(* Logix 5000 project; controller L3 vendor 1 type 14 code 92 rev 20.12; software revision 20.04; part 2 of 9 *)
(* tags used below, declared in another part *)
   B3 : DINT[100];
   CONV_PID_N10_170 : PID;   // *** Tag created for conversion to PID type required for instruction translation ***
   CV_PID_wkk : DINT;
   cv_pmpano : DINT;
   cv_pmprenv : DINT;
   DateTime : DINT[7];   // DINT array tag for retrieve wallclock time through GSV created during conversion
   dbpmpeau : DINT;
   def_ready_pmp_decap_1 : BOOL;
   def_ready_pmp_decap_2 : BOOL;
   def_ready_pmpeau1 : BOOL;
   def_ready_pmpeau2 : BOOL;
   def_ready_ventilo_eau_1 : BOOL;
   def_ready_ventilo_eau_2 : BOOL;
   def_ready_ventilo_eau_3 : BOOL;
   dmd_run_pmp1_decap : BOOL;
   dmd_run_pmp2_decap : BOOL;
   F8 : REAL[100];
   L3_stat : DINT[20];
   limb_pmpeau : DINT;
   limh_pmpeau : DINT;
   N10 : DINT[233];
   N20 : DINT[200];
   N7 : DINT[200];
   N9 : DINT[200];   // niveau decapage vers lancy (n9[10) ;;N9[70]
   ok_arm_io_decap : BOOL;
   okpmpeau1 : BOOL;
   okpmpeau2 : BOOL;
   okventilotour1 : BOOL;
   okventilotour2 : BOOL;
   okventilotour3 : BOOL;
   pid_ANO : PID;
   pid_colmat : PID;
   pid_deg : PID;
   pid_pmpANO : PID;
   pid_pmprenvoi : PID;
   PIDwkk : PID;
   pmpano_inhold : BOOL;
   pmpano_inholdval : DINT;
   pmprenv_inhold : BOOL;
   pmprenv_inholdval : DINT;
   S_bP_dmd_man_pmp_eau : BOOL;
   s_bp_stop_soude : BOOL;
   s_bp_strt_soude : BOOL;
   s_csg_ventilo_ano : DINT;
   S_def_pmp_decap_1 : BOOL;
   S_def_pmp_decap_2 : BOOL;
   S_def_pmpeauano1 : BOOL;
   S_def_pmpeauano2 : BOOL;
   S_def_ventilo_eau1 : BOOL;
   S_def_ventilo_eau2 : BOOL;
   S_def_ventilo_eau3 : BOOL;
   S_FLOW_RETURN_LANCY : DINT;
   S_hiver : BOOL;
   s_nbr_ventilo_ano : DINT;
   S_Q_DEM_NAOH : DINT;
   S_RUN_PMP_DEC1 : BOOL;
   S_RUN_PMP_DEC2 : BOOL;
   S_run_pmpeauano1 : BOOL;
   S_run_pmpeauano2 : BOOL;
   S_run_ventilo_1 : BOOL;
   s_run_ventilo_2 : BOOL;
   S_run_ventilo_3 : BOOL;
   S_SPEED : DINT;
   S_T_ANO : DINT;
   scp_pmp_decap_1 : SCP;
   scp_pmp_decap_2 : SCP;
   scp_ventilo : SCP;
   stat_L3 : DINT[20];
   T4 : TIMER[180];
   T_man_pmp_eau : TIMER;
   T_pmp_decap_1 : TIMER;
   T_pmp_decap_2 : TIMER;
   T_pmpeau_1 : TIMER;
   T_pmpeau_2 : TIMER;
   T_ventilo_eau_1 : TIMER;
   T_ventilo_eau_2 : TIMER;
   T_ventilo_eau_3 : TIMER;
   TIE_PID_wkk : DINT;
   vit_pmp_dec_1 : REAL;
   vit_pmp_dec_2 : DINT;
   vit_renvoi_lancy : DINT;
   vit_ventilo : DINT;
   vitpmpeau : DINT;

PROGRAM _11_PID2   (* main routine _11_PID2 *)

ROUTINE _11_PID2   (* ladder *)
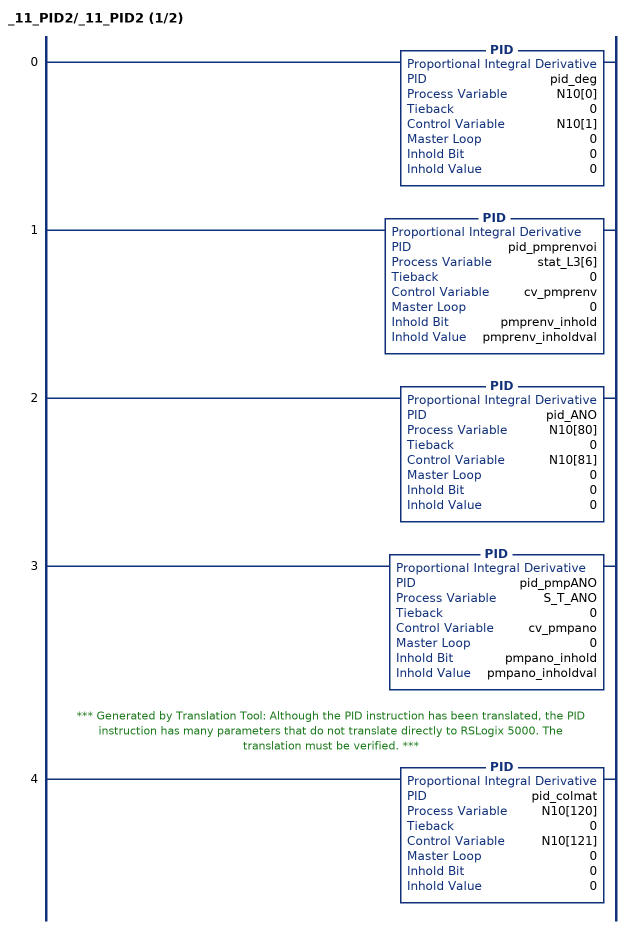
   0: PID(pid_deg,N10[0],0,N10[1],0,0,0);
   1: PID(pid_pmprenvoi,stat_L3[6],0,cv_pmprenv,0,pmprenv_inhold,pmprenv_inholdval);
   2: PID(pid_ANO,N10[80],0,N10[81],0,0,0);
   3: PID(pid_pmpANO,S_T_ANO,0,cv_pmpano,0,pmpano_inhold,pmpano_inholdval);
   // *** Generated by Translation Tool: Although the PID instruction has been translated, the PID instruction has many parameters that do not translate directly to RSLogix 5000. The translation must be verified. ***
   4: PID(pid_colmat,N10[120],0,N10[121],0,0,0);
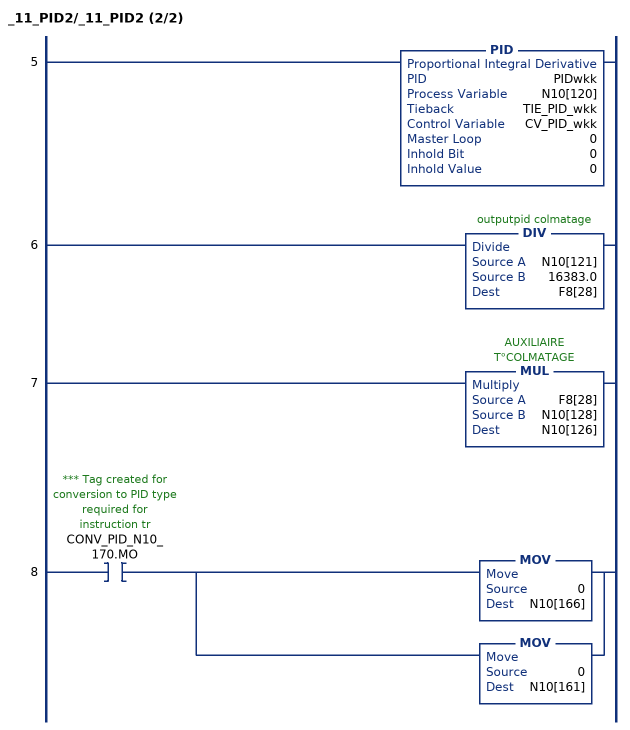
   5: PID(PIDwkk,N10[120],TIE_PID_wkk,CV_PID_wkk,0,0,0);
   6: DIV(N10[121],16383.0,F8[28]);
   7: MUL(F8[28],N10[128],N10[126]);
   8: XIC(CONV_PID_N10_170.MO)[MOV(0,N10[166]) ,MOV(0,N10[161]) ];
END_ROUTINE
END_PROGRAM

PROGRAM _2_GENERAL   (* main routine _2_GENERAL *)

ROUTINE _10_soude_conduct_tour   (* ladder *)
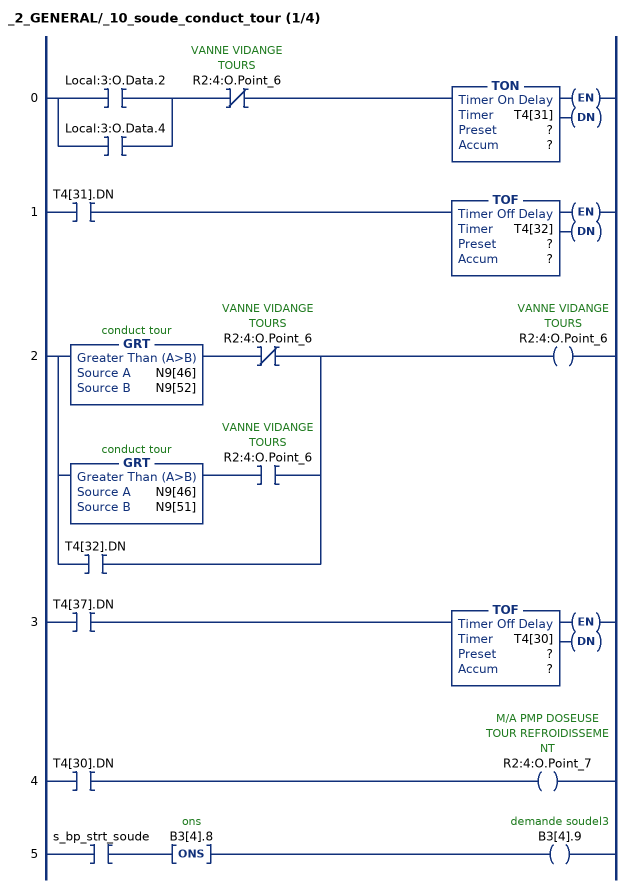
   0: [XIC(Local:3:O.Data.2) ,XIC(Local:3:O.Data.4) ]XIO(R2:4:O.Point_6)TON(T4[31],?,?);
   1: XIC(T4[31].DN)TOF(T4[32],?,?);
   2: [GRT(N9[46],N9[52]) XIO(R2:4:O.Point_6) ,GRT(N9[46],N9[51]) XIC(R2:4:O.Point_6) ,XIC(T4[32].DN) ]OTE(R2:4:O.Point_6);
   3: XIC(T4[37].DN)TOF(T4[30],?,?);
   4: XIC(T4[30].DN)OTE(R2:4:O.Point_7);
   5: XIC(s_bp_strt_soude)ONS(B3[4].8)OTE(B3[4].9);
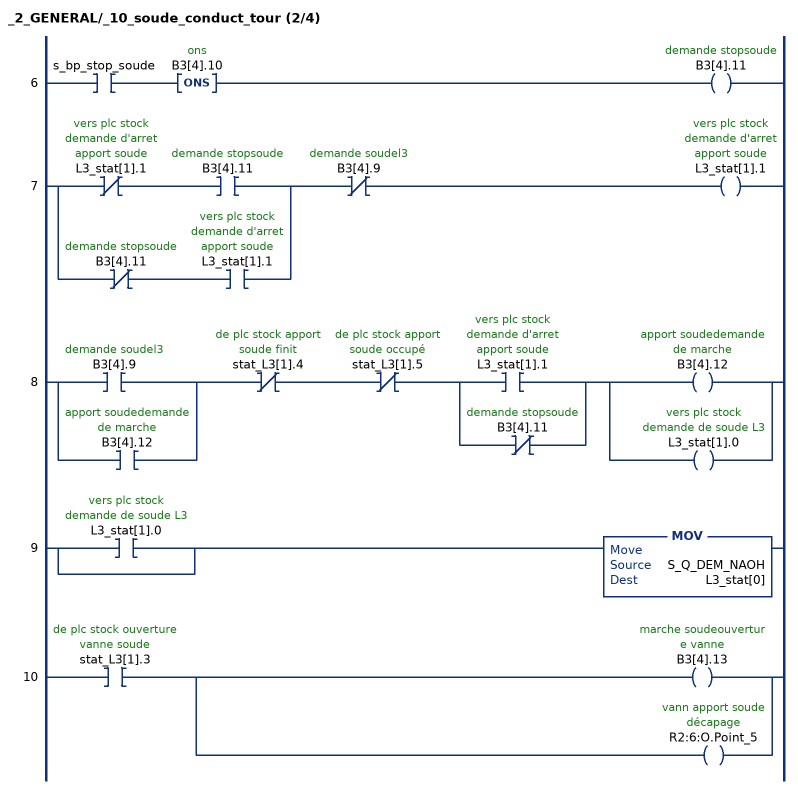
   6: XIC(s_bp_stop_soude)ONS(B3[4].10)OTE(B3[4].11);
   7: [XIO(L3_stat[1].1) XIC(B3[4].11) ,XIO(B3[4].11) XIC(L3_stat[1].1) ]XIO(B3[4].9)OTE(L3_stat[1].1);
   8: [XIC(B3[4].9) ,XIC(B3[4].12) ]XIO(stat_L3[1].4)XIO(stat_L3[1].5)[XIC(L3_stat[1].1) ,XIO(B3[4].11) ][OTE(B3[4].12) ,OTE(L3_stat[1].0) ];
   9: [XIC(L3_stat[1].0) ,]MOV(S_Q_DEM_NAOH,L3_stat[0]);
   10: XIC(stat_L3[1].3)[OTE(B3[4].13) ,OTE(R2:6:O.Point_5) ];
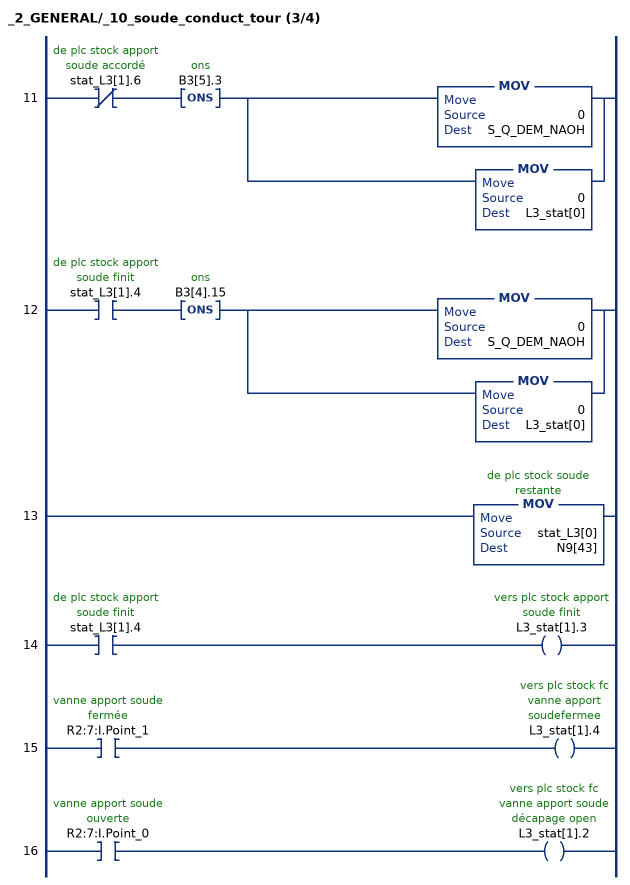
   11: XIO(stat_L3[1].6)ONS(B3[5].3)[MOV(0,S_Q_DEM_NAOH) ,MOV(0,L3_stat[0]) ];
   12: XIC(stat_L3[1].4)ONS(B3[4].15)[MOV(0,S_Q_DEM_NAOH) ,MOV(0,L3_stat[0]) ];
   13: MOV(stat_L3[0],N9[43]);
   14: XIC(stat_L3[1].4)OTE(L3_stat[1].3);
   15: XIC(R2:7:I.Point_1)OTE(L3_stat[1].4);
   16: XIC(R2:7:I.Point_0)OTE(L3_stat[1].2);
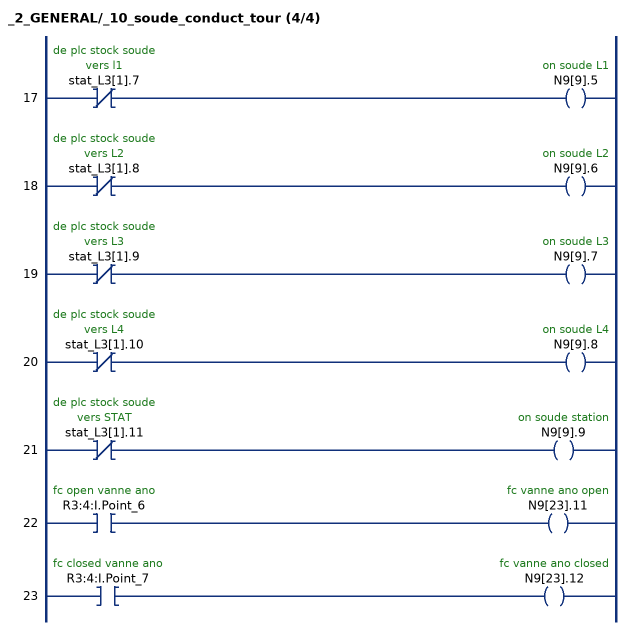
   17: XIO(stat_L3[1].7)OTE(N9[9].5);
   18: XIO(stat_L3[1].8)OTE(N9[9].6);
   19: XIO(stat_L3[1].9)OTE(N9[9].7);
   20: XIO(stat_L3[1].10)OTE(N9[9].8);
   21: XIO(stat_L3[1].11)OTE(N9[9].9);
   22: XIC(R3:4:I.Point_6)OTE(N9[23].11);
   23: XIC(R3:4:I.Point_7)OTE(N9[23].12);
END_ROUTINE

ROUTINE _11_pmp_eau_tour   (* ladder *)
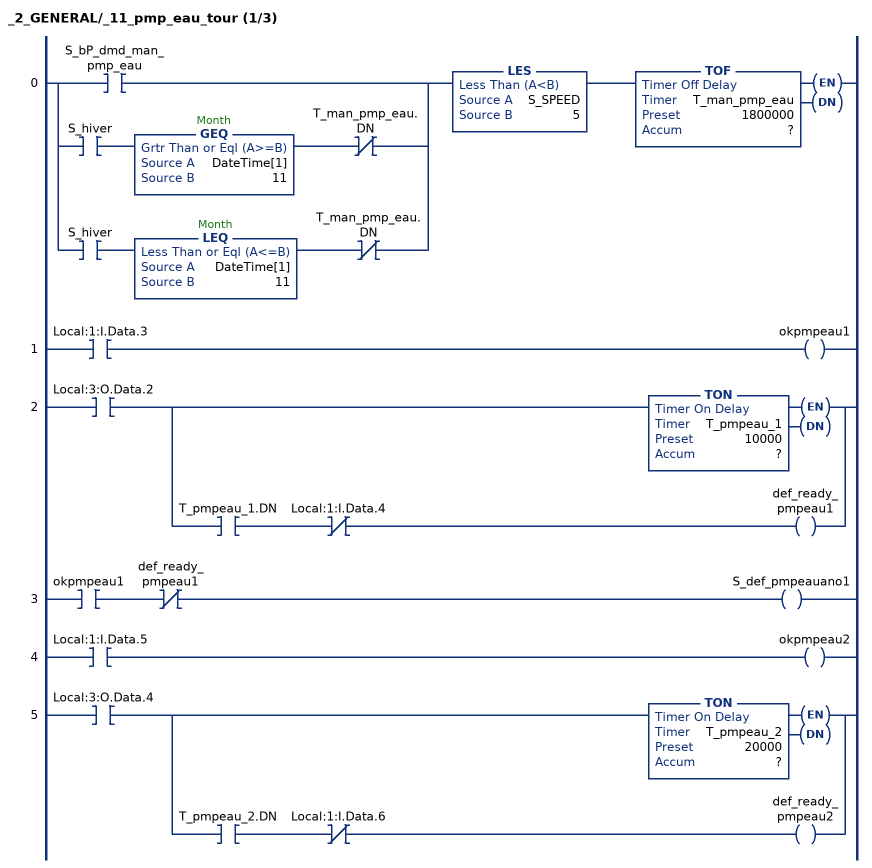
   0: [XIC(S_bP_dmd_man_pmp_eau) ,XIC(S_hiver) GEQ(DateTime[1],11) XIO(T_man_pmp_eau.DN) ,XIC(S_hiver) LEQ(DateTime[1],11) XIO(T_man_pmp_eau.DN) ]LES(S_SPEED,5)TOF(T_man_pmp_eau,?,?);
   1: XIC(Local:1:I.Data.3)OTE(okpmpeau1);
   2: XIC(Local:3:O.Data.2)[TON(T_pmpeau_1,?,?) ,XIC(T_pmpeau_1.DN) XIO(Local:1:I.Data.4) OTE(def_ready_pmpeau1) ];
   3: XIC(okpmpeau1)XIO(def_ready_pmpeau1)OTE(S_def_pmpeauano1);
   4: XIC(Local:1:I.Data.5)OTE(okpmpeau2);
   5: XIC(Local:3:O.Data.4)[TON(T_pmpeau_2,?,?) ,XIC(T_pmpeau_2.DN) XIO(Local:1:I.Data.6) OTE(def_ready_pmpeau2) ];
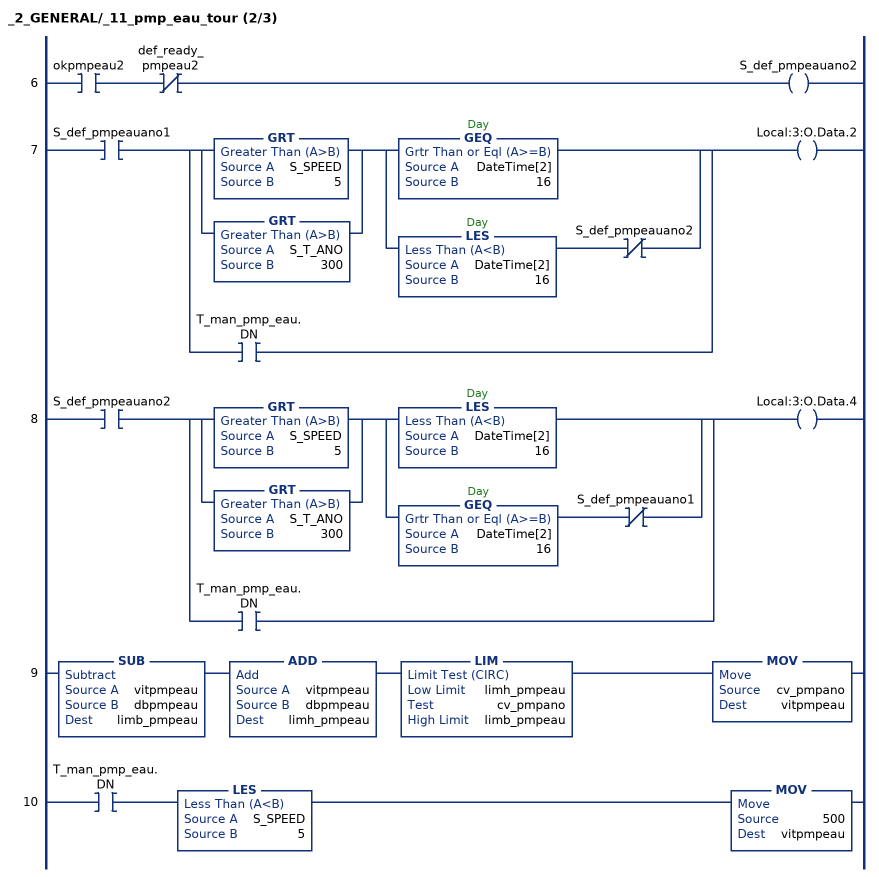
   6: XIC(okpmpeau2)XIO(def_ready_pmpeau2)OTE(S_def_pmpeauano2);
   7: XIC(S_def_pmpeauano1)[[GRT(S_SPEED,5) ,GRT(S_T_ANO,300) ] [GEQ(DateTime[2],16) ,LES(DateTime[2],16) XIO(S_def_pmpeauano2) ] ,XIC(T_man_pmp_eau.DN) ]OTE(Local:3:O.Data.2);
   8: XIC(S_def_pmpeauano2)[[GRT(S_SPEED,5) ,GRT(S_T_ANO,300) ] [LES(DateTime[2],16) ,GEQ(DateTime[2],16) XIO(S_def_pmpeauano1) ] ,XIC(T_man_pmp_eau.DN) ]OTE(Local:3:O.Data.4);
   9: SUB(vitpmpeau,dbpmpeau,limb_pmpeau)ADD(vitpmpeau,dbpmpeau,limh_pmpeau)LIM(limh_pmpeau,cv_pmpano,limb_pmpeau)MOV(cv_pmpano,vitpmpeau);
   10: XIC(T_man_pmp_eau.DN)LES(S_SPEED,5)MOV(500,vitpmpeau);
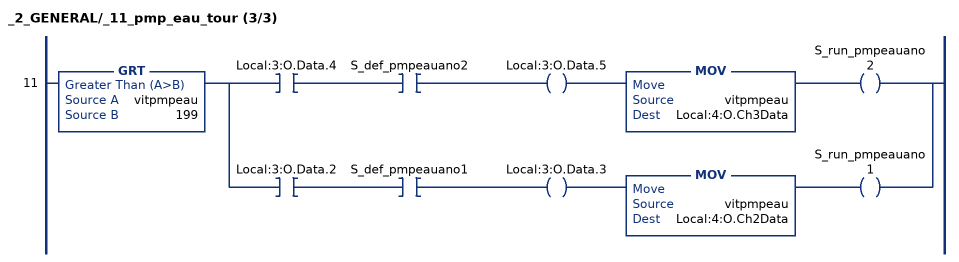
   11: GRT(vitpmpeau,199)[XIC(Local:3:O.Data.4) XIC(S_def_pmpeauano2) OTE(Local:3:O.Data.5) MOV(vitpmpeau,Local:4:O.Ch3Data) OTE(S_run_pmpeauano2) ,XIC(Local:3:O.Data.2) XIC(S_def_pmpeauano1) OTE(Local:3:O.Data.3) MOV(vitpmpeau,Local:4:O.Ch2Data) OTE(S_run_pmpeauano1) ];
END_ROUTINE

ROUTINE _12_ventilo_tour   (* ladder *)
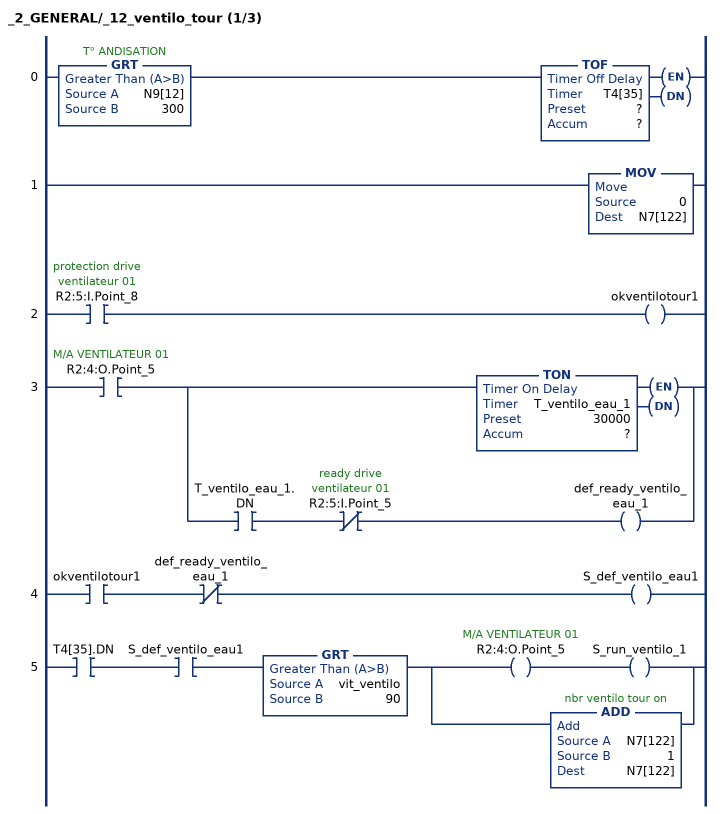
   0: GRT(N9[12],300)TOF(T4[35],?,?);
   1: MOV(0,N7[122]);
   2: XIC(R2:5:I.Point_8)OTE(okventilotour1);
   3: XIC(R2:4:O.Point_5)[TON(T_ventilo_eau_1,?,?) ,XIC(T_ventilo_eau_1.DN) XIO(R2:5:I.Point_5) OTE(def_ready_ventilo_eau_1) ];
   4: XIC(okventilotour1)XIO(def_ready_ventilo_eau_1)OTE(S_def_ventilo_eau1);
   5: XIC(T4[35].DN)XIC(S_def_ventilo_eau1)GRT(vit_ventilo,90)[OTE(R2:4:O.Point_5) OTE(S_run_ventilo_1) ,ADD(N7[122],1,N7[122]) ];
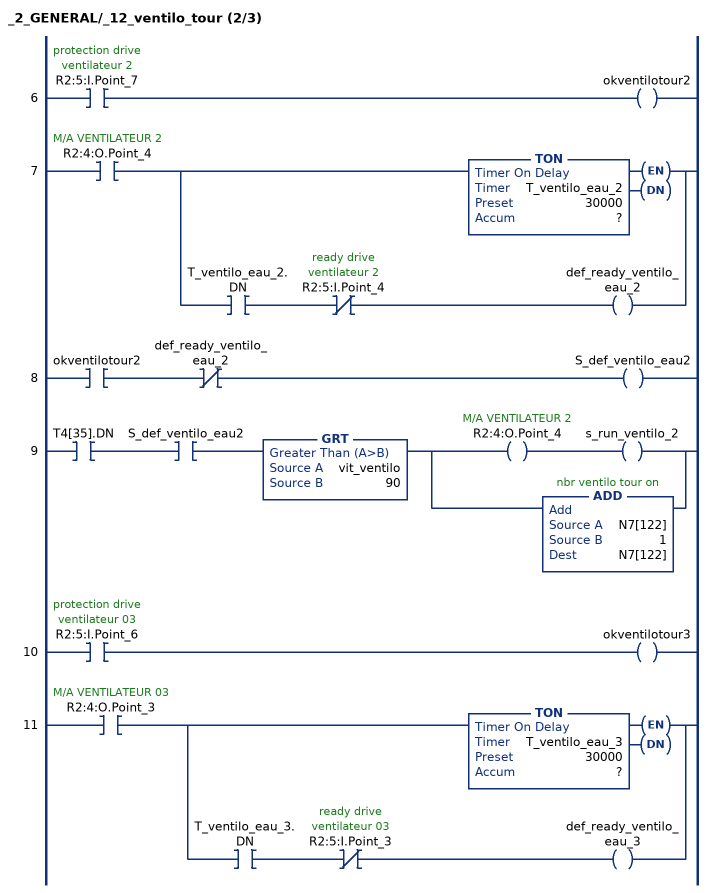
   6: XIC(R2:5:I.Point_7)OTE(okventilotour2);
   7: XIC(R2:4:O.Point_4)[TON(T_ventilo_eau_2,?,?) ,XIC(T_ventilo_eau_2.DN) XIO(R2:5:I.Point_4) OTE(def_ready_ventilo_eau_2) ];
   8: XIC(okventilotour2)XIO(def_ready_ventilo_eau_2)OTE(S_def_ventilo_eau2);
   9: XIC(T4[35].DN)XIC(S_def_ventilo_eau2)GRT(vit_ventilo,90)[OTE(R2:4:O.Point_4) OTE(s_run_ventilo_2) ,ADD(N7[122],1,N7[122]) ];
   10: XIC(R2:5:I.Point_6)OTE(okventilotour3);
   11: XIC(R2:4:O.Point_3)[TON(T_ventilo_eau_3,?,?) ,XIC(T_ventilo_eau_3.DN) XIO(R2:5:I.Point_3) OTE(def_ready_ventilo_eau_3) ];
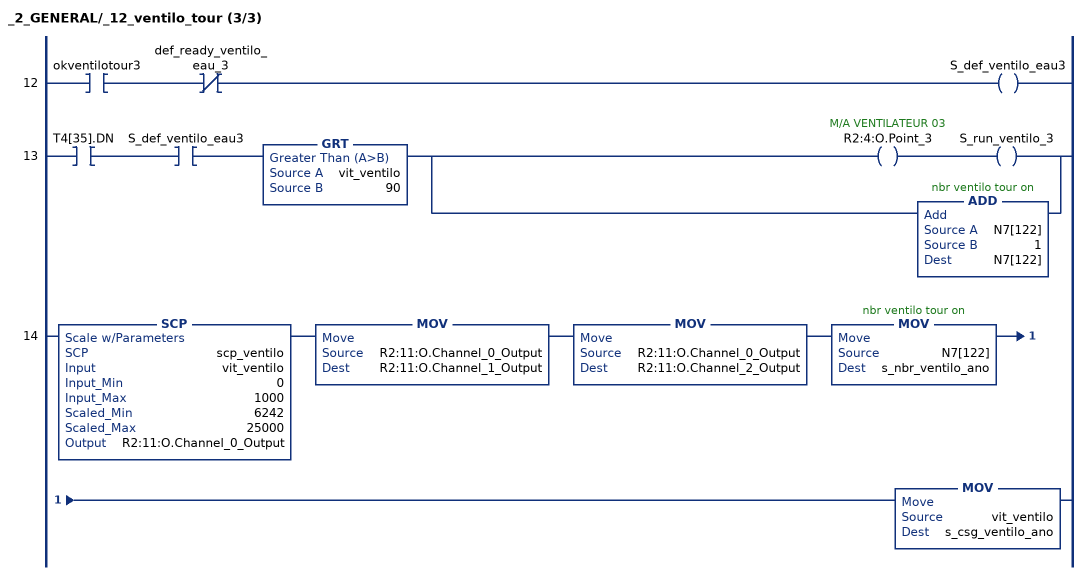
   12: XIC(okventilotour3)XIO(def_ready_ventilo_eau_3)OTE(S_def_ventilo_eau3);
   13: XIC(T4[35].DN)XIC(S_def_ventilo_eau3)GRT(vit_ventilo,90)[OTE(R2:4:O.Point_3) OTE(S_run_ventilo_3) ,ADD(N7[122],1,N7[122]) ];
   14: SCP(scp_ventilo,vit_ventilo,0,1000,6242,25000,R2:11:O.Channel_0_Output)MOV(R2:11:O.Channel_0_Output,R2:11:O.Channel_1_Output)MOV(R2:11:O.Channel_0_Output,R2:11:O.Channel_2_Output)MOV(N7[122],s_nbr_ventilo_ano)MOV(vit_ventilo,s_csg_ventilo_ano);
END_ROUTINE

ROUTINE _13_pmp_decap   (* ladder *)
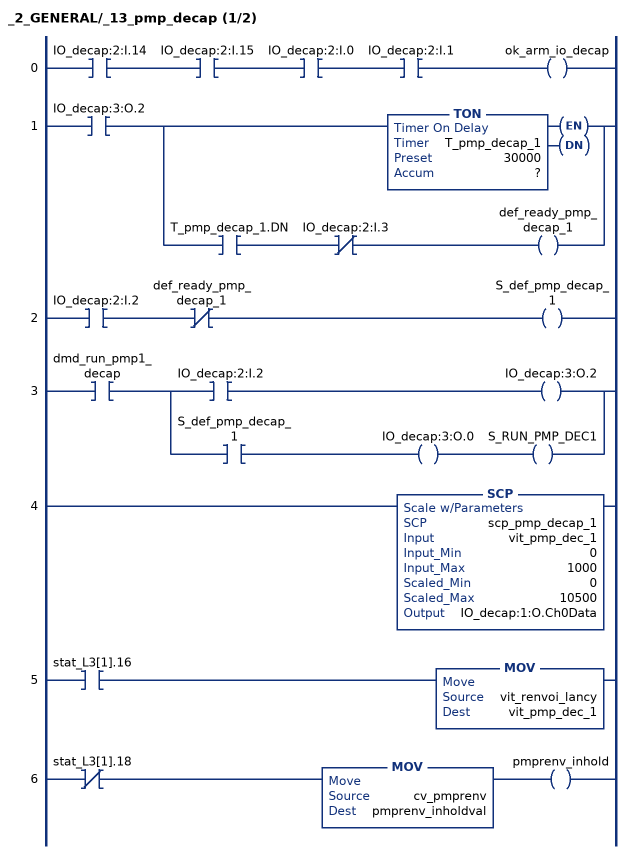
   0: XIC(IO_decap:2:I.14)XIC(IO_decap:2:I.15)XIC(IO_decap:2:I.0)XIC(IO_decap:2:I.1)OTE(ok_arm_io_decap);
   1: XIC(IO_decap:3:O.2)[TON(T_pmp_decap_1,?,?) ,XIC(T_pmp_decap_1.DN) XIO(IO_decap:2:I.3) OTE(def_ready_pmp_decap_1) ];
   2: XIC(IO_decap:2:I.2)XIO(def_ready_pmp_decap_1)OTE(S_def_pmp_decap_1);
   3: XIC(dmd_run_pmp1_decap)[XIC(IO_decap:2:I.2) OTE(IO_decap:3:O.2) ,XIC(S_def_pmp_decap_1) OTE(IO_decap:3:O.0) OTE(S_RUN_PMP_DEC1) ];
   4: SCP(scp_pmp_decap_1,vit_pmp_dec_1,0,1000,0,10500,IO_decap:1:O.Ch0Data);
   5: XIC(stat_L3[1].16)MOV(vit_renvoi_lancy,vit_pmp_dec_1);
   6: XIO(stat_L3[1].18)MOV(cv_pmprenv,pmprenv_inholdval)OTE(pmprenv_inhold);
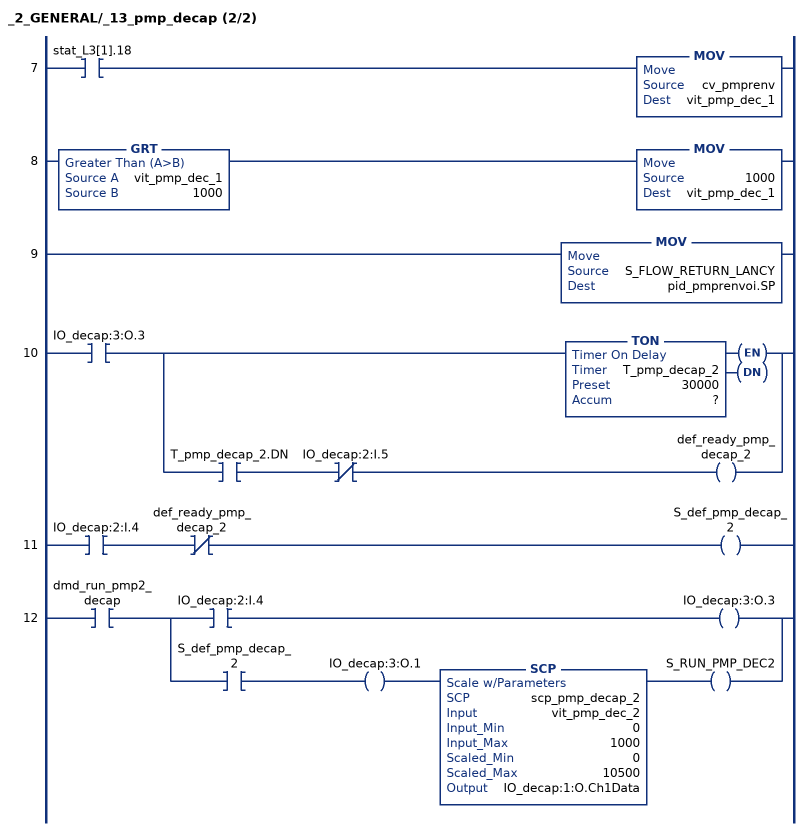
   7: XIC(stat_L3[1].18)MOV(cv_pmprenv,vit_pmp_dec_1);
   8: GRT(vit_pmp_dec_1,1000)MOV(1000,vit_pmp_dec_1);
   9: MOV(S_FLOW_RETURN_LANCY,pid_pmprenvoi.SP);
   10: XIC(IO_decap:3:O.3)[TON(T_pmp_decap_2,?,?) ,XIC(T_pmp_decap_2.DN) XIO(IO_decap:2:I.5) OTE(def_ready_pmp_decap_2) ];
   11: XIC(IO_decap:2:I.4)XIO(def_ready_pmp_decap_2)OTE(S_def_pmp_decap_2);
   12: XIC(dmd_run_pmp2_decap)[XIC(IO_decap:2:I.4) OTE(IO_decap:3:O.3) ,XIC(S_def_pmp_decap_2) OTE(IO_decap:3:O.1) SCP(scp_pmp_decap_2,vit_pmp_dec_2,0,1000,0,10500,IO_decap:1:O.Ch1Data) OTE(S_RUN_PMP_DEC2) ];
END_ROUTINE

ROUTINE _20_ALARM   (* ladder *)
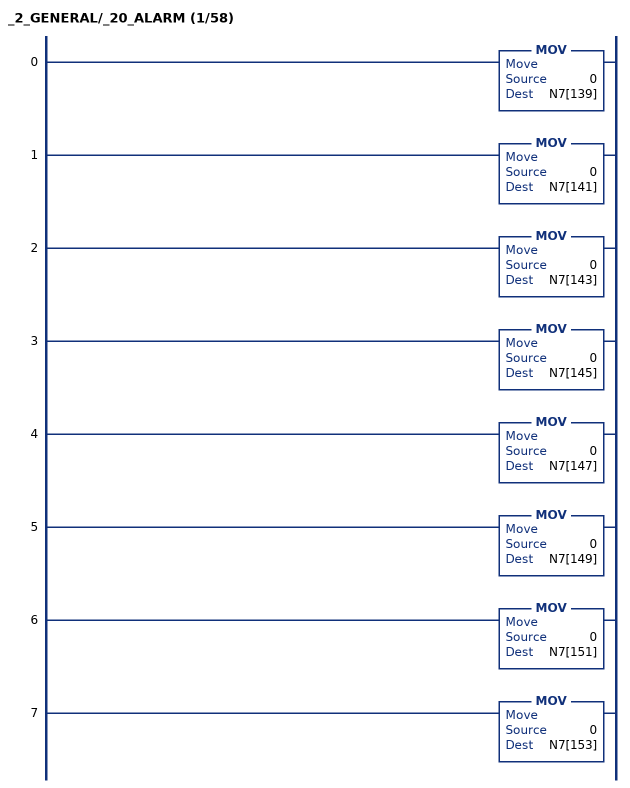
   0: MOV(0,N7[139]);
   1: MOV(0,N7[141]);
   2: MOV(0,N7[143]);
   3: MOV(0,N7[145]);
   4: MOV(0,N7[147]);
   5: MOV(0,N7[149]);
   6: MOV(0,N7[151]);
   7: MOV(0,N7[153]);
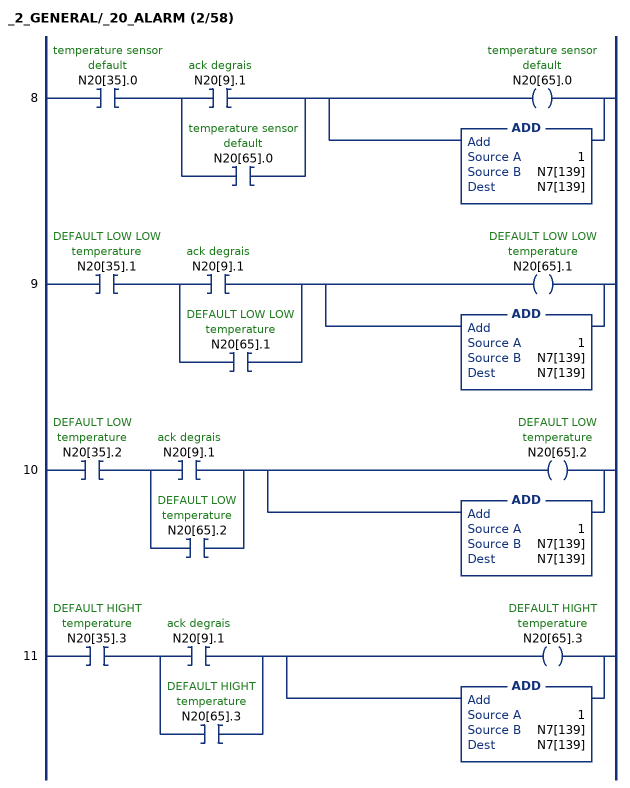
   8: XIC(N20[35].0)[XIC(N20[9].1) ,XIC(N20[65].0) ][OTE(N20[65].0) ,ADD(1,N7[139],N7[139]) ];
   9: XIC(N20[35].1)[XIC(N20[9].1) ,XIC(N20[65].1) ][OTE(N20[65].1) ,ADD(1,N7[139],N7[139]) ];
   10: XIC(N20[35].2)[XIC(N20[9].1) ,XIC(N20[65].2) ][OTE(N20[65].2) ,ADD(1,N7[139],N7[139]) ];
   11: XIC(N20[35].3)[XIC(N20[9].1) ,XIC(N20[65].3) ][OTE(N20[65].3) ,ADD(1,N7[139],N7[139]) ];
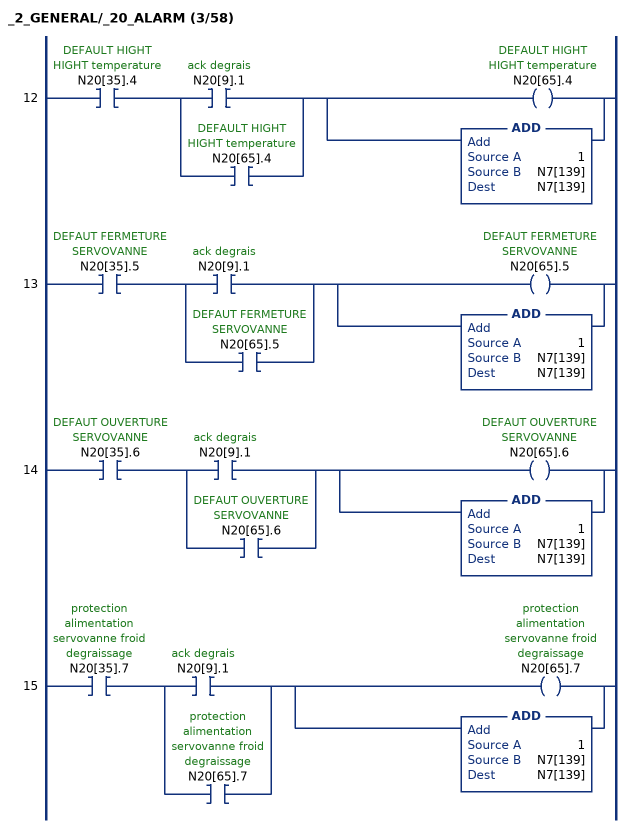
   12: XIC(N20[35].4)[XIC(N20[9].1) ,XIC(N20[65].4) ][OTE(N20[65].4) ,ADD(1,N7[139],N7[139]) ];
   13: XIC(N20[35].5)[XIC(N20[9].1) ,XIC(N20[65].5) ][OTE(N20[65].5) ,ADD(1,N7[139],N7[139]) ];
   14: XIC(N20[35].6)[XIC(N20[9].1) ,XIC(N20[65].6) ][OTE(N20[65].6) ,ADD(1,N7[139],N7[139]) ];
   15: XIC(N20[35].7)[XIC(N20[9].1) ,XIC(N20[65].7) ][OTE(N20[65].7) ,ADD(1,N7[139],N7[139]) ];
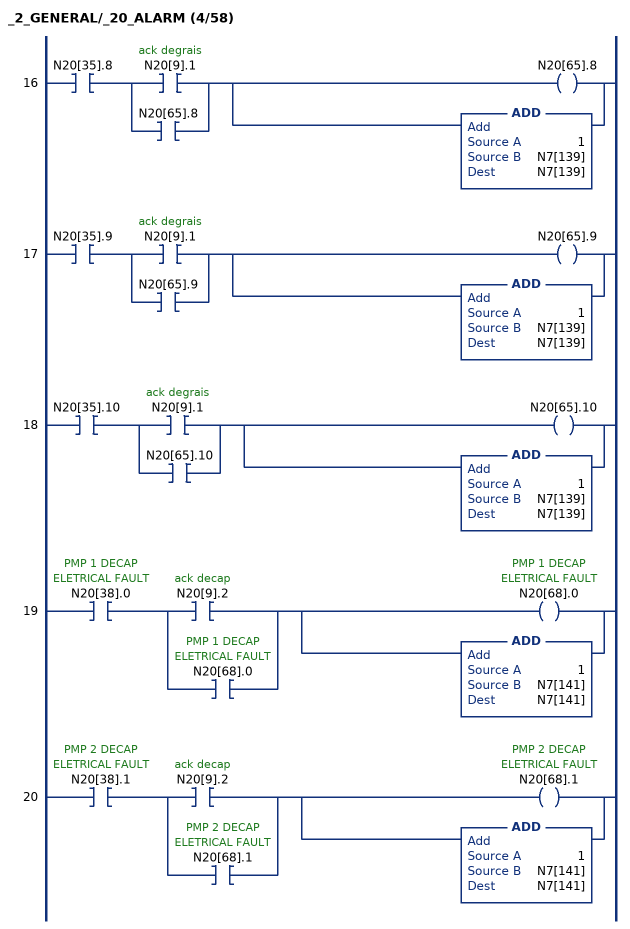
   16: XIC(N20[35].8)[XIC(N20[9].1) ,XIC(N20[65].8) ][OTE(N20[65].8) ,ADD(1,N7[139],N7[139]) ];
   17: XIC(N20[35].9)[XIC(N20[9].1) ,XIC(N20[65].9) ][OTE(N20[65].9) ,ADD(1,N7[139],N7[139]) ];
   18: XIC(N20[35].10)[XIC(N20[9].1) ,XIC(N20[65].10) ][OTE(N20[65].10) ,ADD(1,N7[139],N7[139]) ];
   19: XIC(N20[38].0)[XIC(N20[9].2) ,XIC(N20[68].0) ][OTE(N20[68].0) ,ADD(1,N7[141],N7[141]) ];
   20: XIC(N20[38].1)[XIC(N20[9].2) ,XIC(N20[68].1) ][OTE(N20[68].1) ,ADD(1,N7[141],N7[141]) ];
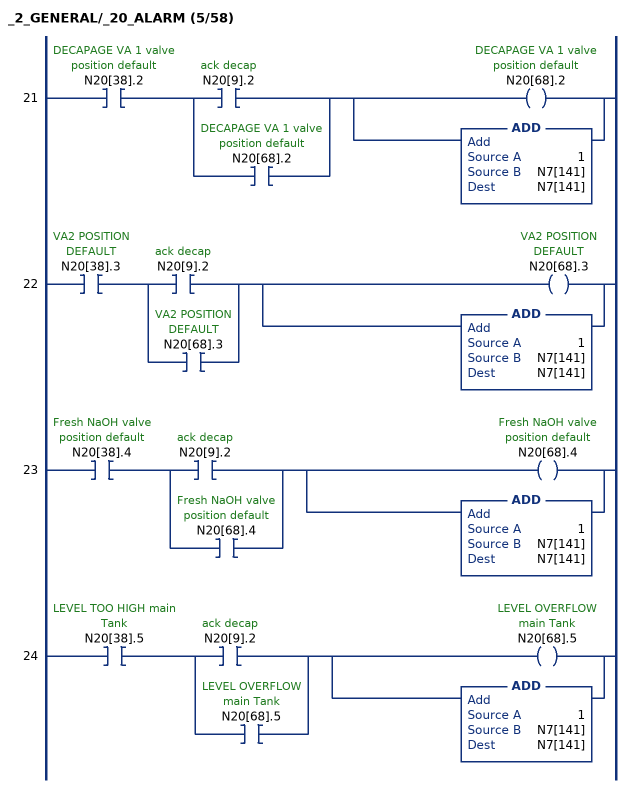
   21: XIC(N20[38].2)[XIC(N20[9].2) ,XIC(N20[68].2) ][OTE(N20[68].2) ,ADD(1,N7[141],N7[141]) ];
   22: XIC(N20[38].3)[XIC(N20[9].2) ,XIC(N20[68].3) ][OTE(N20[68].3) ,ADD(1,N7[141],N7[141]) ];
   23: XIC(N20[38].4)[XIC(N20[9].2) ,XIC(N20[68].4) ][OTE(N20[68].4) ,ADD(1,N7[141],N7[141]) ];
   24: XIC(N20[38].5)[XIC(N20[9].2) ,XIC(N20[68].5) ][OTE(N20[68].5) ,ADD(1,N7[141],N7[141]) ];
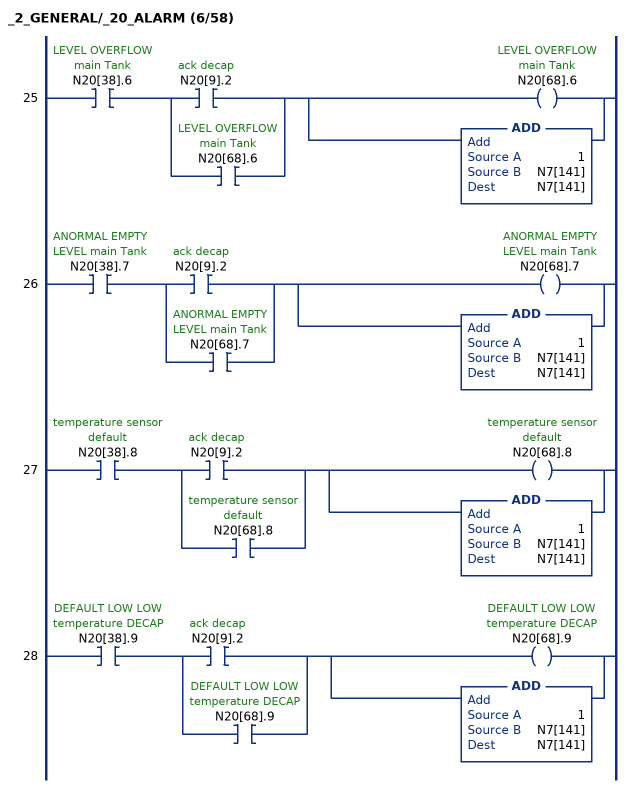
   25: XIC(N20[38].6)[XIC(N20[9].2) ,XIC(N20[68].6) ][OTE(N20[68].6) ,ADD(1,N7[141],N7[141]) ];
   26: XIC(N20[38].7)[XIC(N20[9].2) ,XIC(N20[68].7) ][OTE(N20[68].7) ,ADD(1,N7[141],N7[141]) ];
   27: XIC(N20[38].8)[XIC(N20[9].2) ,XIC(N20[68].8) ][OTE(N20[68].8) ,ADD(1,N7[141],N7[141]) ];
   28: XIC(N20[38].9)[XIC(N20[9].2) ,XIC(N20[68].9) ][OTE(N20[68].9) ,ADD(1,N7[141],N7[141]) ];
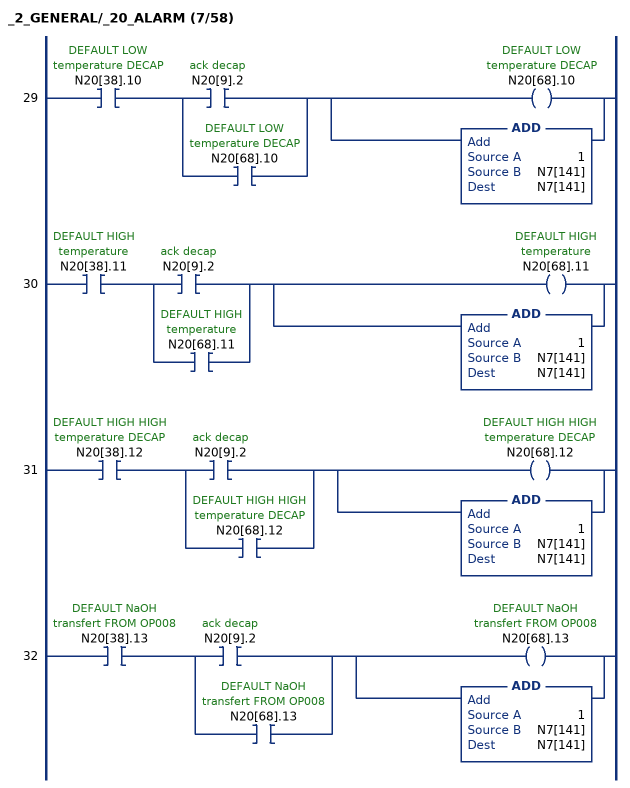
   29: XIC(N20[38].10)[XIC(N20[9].2) ,XIC(N20[68].10) ][OTE(N20[68].10) ,ADD(1,N7[141],N7[141]) ];
   30: XIC(N20[38].11)[XIC(N20[9].2) ,XIC(N20[68].11) ][OTE(N20[68].11) ,ADD(1,N7[141],N7[141]) ];
   31: XIC(N20[38].12)[XIC(N20[9].2) ,XIC(N20[68].12) ][OTE(N20[68].12) ,ADD(1,N7[141],N7[141]) ];
   32: XIC(N20[38].13)[XIC(N20[9].2) ,XIC(N20[68].13) ][OTE(N20[68].13) ,ADD(1,N7[141],N7[141]) ];
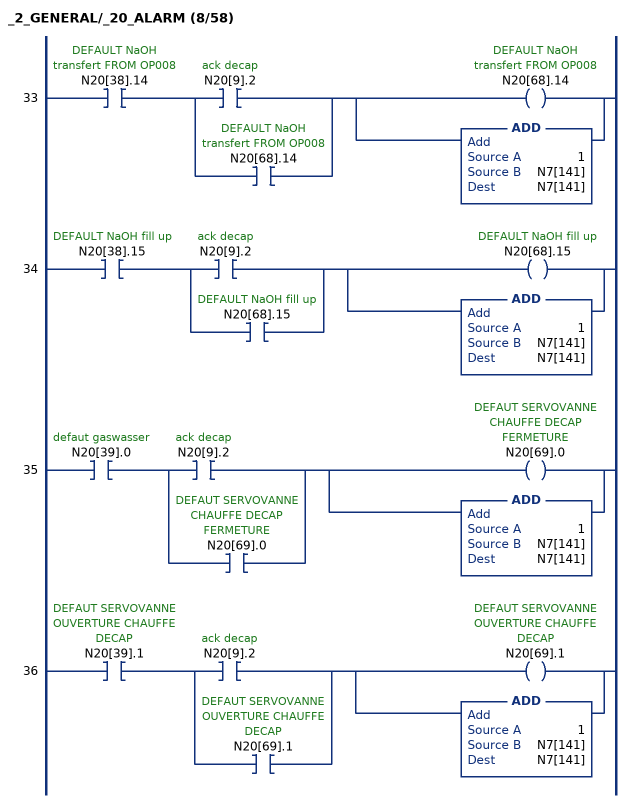
   33: XIC(N20[38].14)[XIC(N20[9].2) ,XIC(N20[68].14) ][OTE(N20[68].14) ,ADD(1,N7[141],N7[141]) ];
   34: XIC(N20[38].15)[XIC(N20[9].2) ,XIC(N20[68].15) ][OTE(N20[68].15) ,ADD(1,N7[141],N7[141]) ];
   35: XIC(N20[39].0)[XIC(N20[9].2) ,XIC(N20[69].0) ][OTE(N20[69].0) ,ADD(1,N7[141],N7[141]) ];
   36: XIC(N20[39].1)[XIC(N20[9].2) ,XIC(N20[69].1) ][OTE(N20[69].1) ,ADD(1,N7[141],N7[141]) ];
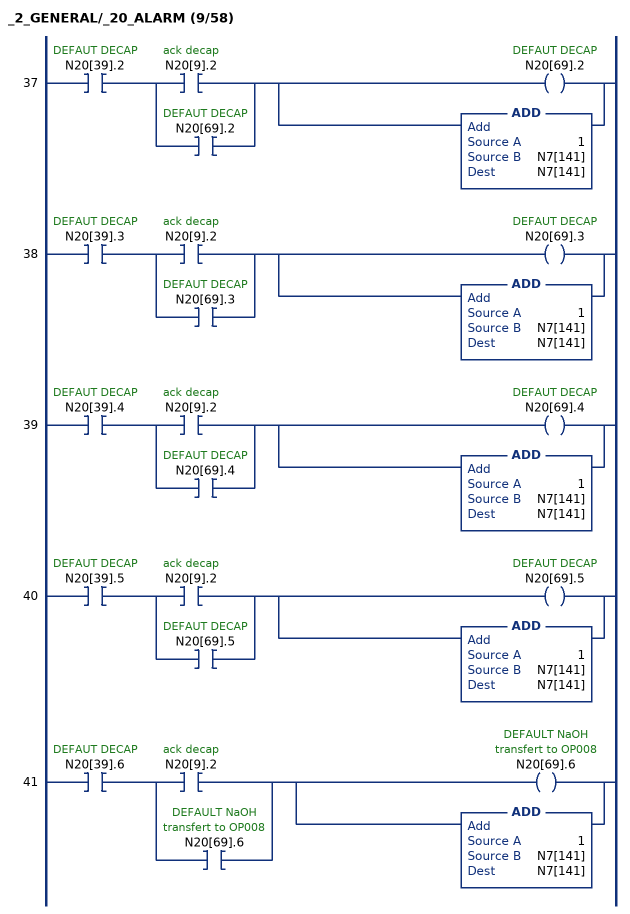
   37: XIC(N20[39].2)[XIC(N20[9].2) ,XIC(N20[69].2) ][OTE(N20[69].2) ,ADD(1,N7[141],N7[141]) ];
   38: XIC(N20[39].3)[XIC(N20[9].2) ,XIC(N20[69].3) ][OTE(N20[69].3) ,ADD(1,N7[141],N7[141]) ];
   39: XIC(N20[39].4)[XIC(N20[9].2) ,XIC(N20[69].4) ][OTE(N20[69].4) ,ADD(1,N7[141],N7[141]) ];
   40: XIC(N20[39].5)[XIC(N20[9].2) ,XIC(N20[69].5) ][OTE(N20[69].5) ,ADD(1,N7[141],N7[141]) ];
   41: XIC(N20[39].6)[XIC(N20[9].2) ,XIC(N20[69].6) ][OTE(N20[69].6) ,ADD(1,N7[141],N7[141]) ];
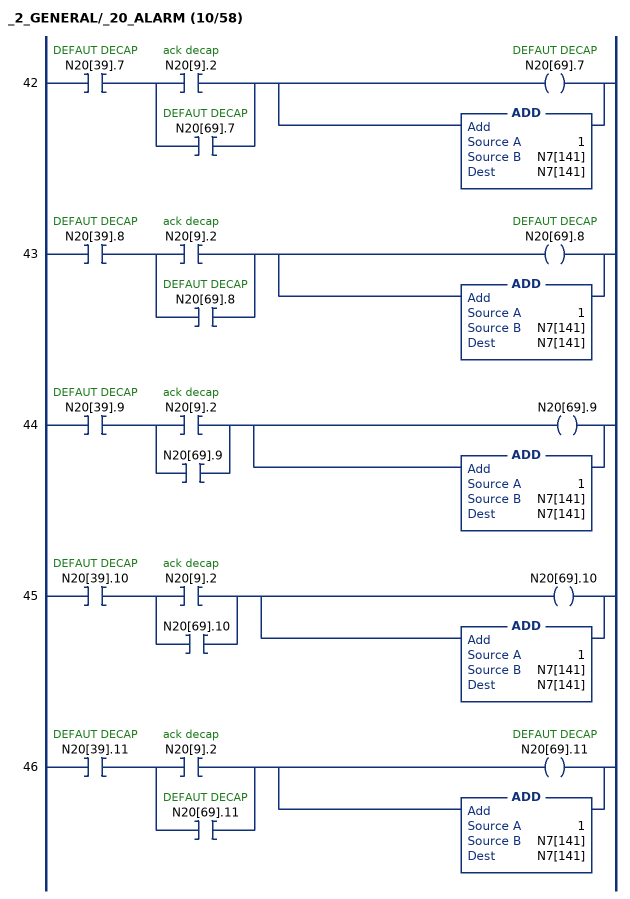
   42: XIC(N20[39].7)[XIC(N20[9].2) ,XIC(N20[69].7) ][OTE(N20[69].7) ,ADD(1,N7[141],N7[141]) ];
   43: XIC(N20[39].8)[XIC(N20[9].2) ,XIC(N20[69].8) ][OTE(N20[69].8) ,ADD(1,N7[141],N7[141]) ];
   44: XIC(N20[39].9)[XIC(N20[9].2) ,XIC(N20[69].9) ][OTE(N20[69].9) ,ADD(1,N7[141],N7[141]) ];
   45: XIC(N20[39].10)[XIC(N20[9].2) ,XIC(N20[69].10) ][OTE(N20[69].10) ,ADD(1,N7[141],N7[141]) ];
   46: XIC(N20[39].11)[XIC(N20[9].2) ,XIC(N20[69].11) ][OTE(N20[69].11) ,ADD(1,N7[141],N7[141]) ];
